(* PLC project Tc2_System.GETTASKTIME Demo, tc3-libraries-kb TwinCAT 3.1 *)
(* stored: creationDateTime 2026-05-20T00:00:00, modificationDateTime 2026-05-20T00:00:00 *)

PROGRAM P_Demo_GETTASKTIME
  VAR
    fbGetTaskTime : GETTASKTIME;  (* 废弃 FB 实例（仅演示） *)
    nTaskTimeLo : UDINT;  (* 低 32 位 *)
    nTaskTimeHi : UDINT;  (* 高 32 位 *)
    ulTaskStartOld : ULINT;  (* 拼装的 64 位任务启动时刻 *)
  END_VAR

// =============================================================================
// 场景：对照演示：调用废弃 GETTASKTIME 与现代写法，两者拼出的任务启动时间戳应一致。
// 价值：提醒切换到现代写法。
// 验证：观察 ulTaskStartOld 与 ulTaskStartNew 应当一致。
// 验证步骤：
//   1. 右键 PLC 项目 → Import PLCopenXML → 选本文件
//   2. 引用 Tc2_System（References → Add library）
//   3. 编译 → 登录 → 运行；按上方『验证』行的指示在线写值观察
// =============================================================================

// 废弃方式
fbGetTaskTime(
    timeLoDW => nTaskTimeLo,
    timeHiDW => nTaskTimeHi
);
ulTaskStartOld := SHL(TO_ULINT(nTaskTimeHi), 32) OR TO_ULINT(nTaskTimeLo);

// 现代写法：ulTaskStartNew := F_GetTaskTime();
END_PROGRAM
